TYPE (* ButtonActivationCode Struct *)
  (* Version 1.0, 2025-07-21, franz *)
  ButtonActivationCode_S : STRUCT
    code : USINT := 255;
    bCyclic : BOOL := FALSE;
  END_STRUCT;
END_TYPE
